// SIMATIC S7-200 project (STEP 7-Micro/WIN), CPU 221 REL 01.10

SYMBOL_TABLE USR1
Store_POT0       MW0      // The value at POT0 is stored in this memory word.
Old_POT0         MW2      // The previous value at POT0 is stored in this memory word
Always_On        SM0.0    // This bit is always on.
First_Scan_On    SM0.1    // This bit is on for the first scan cycle only.
POT0_Value       SMB28    // Stores value entered by analog adjustment 0. Updated once per cycle in STOP/RUN
PLS0_Ctrl        SMB67    // Controls pulse train output & pulse width modulation functions for output Q0.0.
PLS0_Cycle       SMW68    // Cycle time value, pulse train or pls. width modulation output 0. SMB68 is MSB.
PWM0_PW          SMW70    // Pulse width value of pulse width modulation output 0. SMB70 is the MSB.
END_SYMBOL_TABLE

ORGANIZATION_BLOCK MAIN:OB1
TITLE= 题目：灯泡亮度控制
// ***概述***
// 这个示例解释了一个使用S7-200的集成高速脉冲输出指令来控制灯泡(24V/1W)
// 亮度的例子，模拟电位器0的设置值影响输出端Q0.0方波信号的脉冲宽度，也就
// 是灯泡的亮度。调整电位器时需要一把(2.5mm)螺丝刀。
// ***程序和注释***
// 在程序的每次扫描过程中，模拟电位器0的值，通过特殊存储字节SMB28被拷贝到内存
// 字MW0的低字节MB1。电位器的值除以8作为脉宽，脉宽和脉冲周期的比率大致决定了灯
// 泡的亮度(相对于最大亮度)。除以8会带来这样一个额外的好处，即丢弃了SMB28所存
// 值的3个最低有效位，从而使程序更稳定。如果电位器值变化了，那么将重新初始化
// 输出端Q0.0的脉宽调制，借此电位器的新值将被变换成脉宽的毫秒值。
//    例：SMB28=80  (电位器0的值)
//        80/8=10
//        10/25(=脉宽/周期)=40%(电压时间比)=40%最大亮度
// 标题：用电位器调灯泡亮度
// 
BEGIN
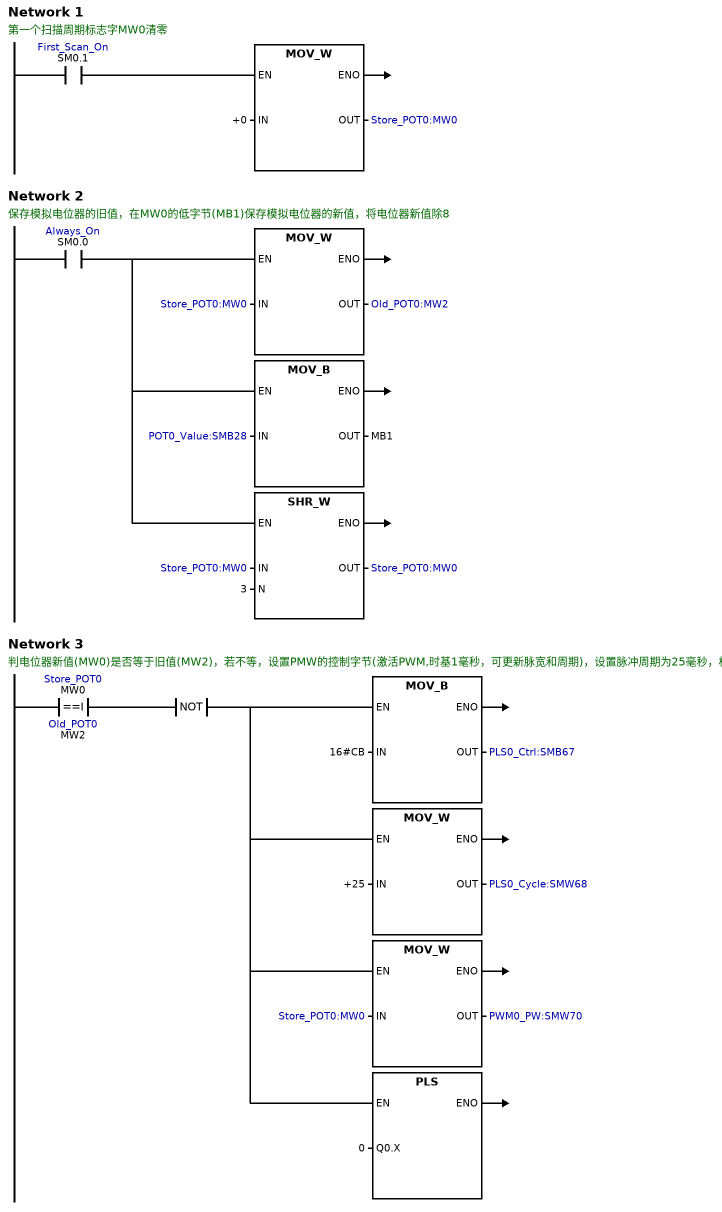
Network 1
// 第一个扫描周期标志字MW0清零
// 第一次扫描SM0.1=1
// 标志字MW0清零
LD     First_Scan_On:SM0.1
MOVW   +0, Store_POT0:MW0
Network 2
// 保存模拟电位器的旧值，在MW0的低字节(MB1)保存模拟电位器的新值，将电位器新值除8
//设置栈顶(SM0.0总是1)
// 保存电位器的旧值
// 在MW0的低字节(MB1)保存模拟电位器新值
// 将电位器新值除8
LD     Always_On:SM0.0
MOVW   Store_POT0:MW0, Old_POT0:MW2
MOVB   POT0_Value:SMB28, MB1
SRW    Store_POT0:MW0, 3
Network 3
// 判电位器新值(MW0)是否等于旧值(MW2)，若不等，设置PMW的控制字节(激活PWM,时基1毫秒，可更新脉宽和周期)，设置脉冲周期为25毫秒，根据电位器值设置脉宽。
// 输出端Q0.0输出脉宽
// 判电位器新值(MW0)是否等于旧值(MW2)
// 若不等
// 设置PMW的控制字节(激活PWM,时基1毫秒，
//可更新脉宽和周期)
//设置脉冲周期为25毫秒
// 根据电位器值设置脉宽。
// 在输出端Q0.0输出脉宽
LDW=   Store_POT0:MW0, Old_POT0:MW2
NOT
MOVB   16#CB, PLS0_Ctrl:SMB67
MOVW   +25, PLS0_Cycle:SMW68
MOVW   Store_POT0:MW0, PWM0_PW:SMW70
PLS    0
Network 4 //  主程序结束
// MEND					
// 
END_ORGANIZATION_BLOCK
